//==================================================================================================
//								RJM Maszyny sp. z o.o.
//									04.02.2022
//	Sterowanie cewką
// 	v1.0	|| TC v 3.1.4024.22		|| - pierwsza wersja
//==================================================================================================
FUNCTION_BLOCK FB_ElektrozaworCewka
VAR
	Wyjscie							AT %Q*	: BOOL;
END_VAR

//==================================================================================================
//								RJM Maszyny sp. z o.o.
//									13.05.2022
//	Włączenie cewki
// 	v1.0	|| TC v 3.1.4024.22		|| - pierwsza wersja
//==================================================================================================
METHOD Wlacz : BOOL
VAR_INPUT
END_VAR
Wyjscie										:= TRUE;
END_METHOD

//==================================================================================================
//								RJM Maszyny sp. z o.o.
//									13.05.2022
//	Wyłączenie cewki
// 	v1.0	|| TC v 3.1.4024.22		|| - pierwsza wersja
//==================================================================================================
METHOD Wylacz : BOOL
VAR_INPUT
END_VAR
Wyjscie										:= FALSE;
END_METHOD

END_FUNCTION_BLOCK

(* stored: Version 1.1.0.1, ProductVersion 3.1.4024.11
   POU FB_ElektrozaworCewka: Id {606fac5f-70dc-43dc-8167-f3c1b1aef47c}, SpecialFunc None
   Method Wlacz: Id {eff36729-b228-4a55-8531-e9f160274bea}
   Method Wylacz: Id {b1ce8405-f55e-4e13-85a7-457bea2892cd} *)
